{attribute 'GeneratedUsingTerminal: EK1100-0000-0018'}
{attribute addProperty BoxType "EK1100-0000-0018"}
{attribute addProperty Id "Beckhoff_EKM1xxxEK1122Beckhoff_EKM1xxxEK1122_63323493372"}
{attribute addProperty CRC "294761938"}
{attribute addProperty Size "372"}
TYPE Beckhoff_EKM1xxx_1191B5D2 EXTENDS EK1100_1FC0878B :
STRUCT
	{attribute addProperty Name "Beckhoff_EKM1xxxEK1122"}
	{attribute addProperty PreviousPort "Beckhoff EKM1xxx : B"}
	Beckhoff_EKM1xxxEK1122 : Beckhoff_EKM1xxxEK1122_63323493;
END_STRUCT
END_TYPE

(* stored: Version 1.2.0.0, ProductVersion 3.1.4024.9
   DUT Beckhoff_EKM1xxx_1191B5D2: Id {db413de7-dd0f-4864-a293-7519750e61f4} *)
